INTERFACE I_VolumeFlowSensor

PROPERTY VolumeFlow : REAL
GET
END_GET
END_PROPERTY

END_INTERFACE

(* stored: Version 1.1.0.1
   Itf I_VolumeFlowSensor: Id {788adee9-3c81-47b7-b107-04763dfb9584}
   Property VolumeFlow: Id {2727b38c-5799-4eb9-981c-4bb8da8fa637}
   Get Get: Id {c8a4b2b1-839f-4831-96e7-c9001554f03c} *)
